SUBAPPLICATION Uebung_032 (* LED Strip Blinkende LED *)
  (* Standard: 61499-2; Description: Copyright (c) 2023 Meisterschulen am Ostbahnhof This program and the accompanying materials are made available under the terms of the Eclipse Public License 2.0 which is available at https://www.eclipse.org/legal/epl-2.0/ SPDX-License-Identifier: EPL-2.0 *)
  (* Version 1.0, 2023-10-23, Franz Höpfinger, Meisterschulen am Ostbahnhof, initial API and implementation and/or initial documentation *)
  PACKAGE Uebungen;
  IMPORT logiBUS::io::DI::logiBUS_DI::Input_I1;
  IMPORT logiBUS::io::DI::logiBUS_DI::Input_I2;
  IMPORT logiBUS::io::DI::logiBUS_DI::Input_I3;
  IMPORT logiBUS::io::DI::logiBUS_DI::Input_I4;
  IMPORT logiBUS::io::DO_LED::LED_COLOURS;
  IMPORT logiBUS::io::DO_LED::LED_FREQ;
  IMPORT logiBUS::io::DO_LED::LED_strip;
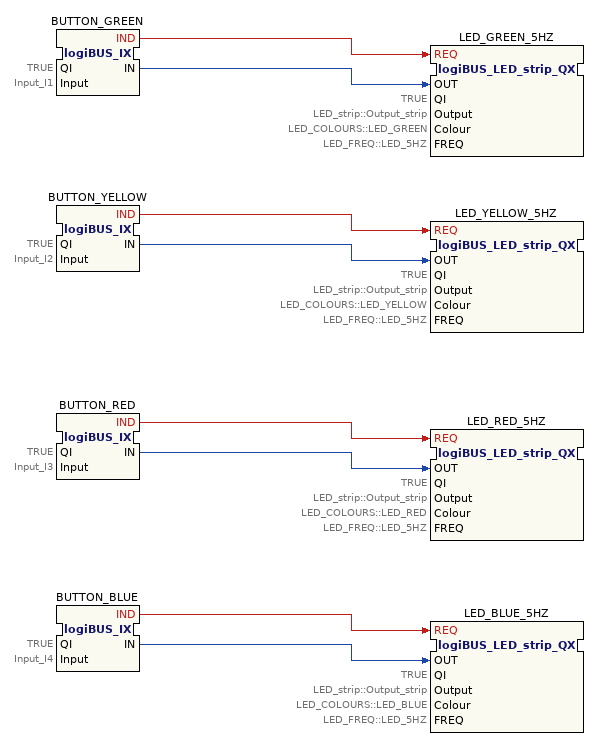
  FBS
    LED_GREEN_5HZ : logiBUS::io::DO_LED::logiBUS_LED_strip_QX(QI := TRUE, Output := LED_strip::Output_strip, Colour := LED_COLOURS::LED_GREEN, FREQ := LED_FREQ::LED_5HZ);
    BUTTON_GREEN : logiBUS::io::DI::logiBUS_IX(QI := TRUE, Input := Input_I1);
    BUTTON_YELLOW : logiBUS::io::DI::logiBUS_IX(QI := TRUE, Input := Input_I2);
    LED_YELLOW_5HZ : logiBUS::io::DO_LED::logiBUS_LED_strip_QX(QI := TRUE, Output := LED_strip::Output_strip, Colour := LED_COLOURS::LED_YELLOW, FREQ := LED_FREQ::LED_5HZ);
    BUTTON_RED : logiBUS::io::DI::logiBUS_IX(QI := TRUE, Input := Input_I3);
    LED_RED_5HZ : logiBUS::io::DO_LED::logiBUS_LED_strip_QX(QI := TRUE, Output := LED_strip::Output_strip, Colour := LED_COLOURS::LED_RED, FREQ := LED_FREQ::LED_5HZ);
    BUTTON_BLUE : logiBUS::io::DI::logiBUS_IX(QI := TRUE, Input := Input_I4);
    LED_BLUE_5HZ : logiBUS::io::DO_LED::logiBUS_LED_strip_QX(QI := TRUE, Output := LED_strip::Output_strip, Colour := LED_COLOURS::LED_BLUE, FREQ := LED_FREQ::LED_5HZ);
  END_FBS
  EVENT_CONNECTIONS
    BUTTON_GREEN.IND TO LED_GREEN_5HZ.REQ;
    BUTTON_YELLOW.IND TO LED_YELLOW_5HZ.REQ;
    BUTTON_RED.IND TO LED_RED_5HZ.REQ;
    BUTTON_BLUE.IND TO LED_BLUE_5HZ.REQ;
  END_CONNECTIONS
  DATA_CONNECTIONS
    BUTTON_GREEN.IN TO LED_GREEN_5HZ.OUT;
    BUTTON_YELLOW.IN TO LED_YELLOW_5HZ.OUT;
    BUTTON_RED.IN TO LED_RED_5HZ.OUT;
    BUTTON_BLUE.IN TO LED_BLUE_5HZ.OUT;
  END_CONNECTIONS
END_SUBAPPLICATION
